FUNCTION_BLOCK Ref_ramp
VAR_INPUT
	Speed_req:INT;
	Allowed_speed:INT;
	Rate:INT;
	Zero:BOOL;
	S_Func_scans:INT;
END_VAR
VAR_OUTPUT
	Speed_ref:INT;
END_VAR
VAR
	Speed_req_real: REAL;
	Speed_step: REAL;
	Speed_ref_real: REAL;
	Speed_up: BOOL;
END_VAR
VAR // added by the converter: edge detectors and wires of the graphical bodies
    _w1, _w2, _w4, _w5, _w6, _w7, _w9, _w10 : ANY;
    _w3 : BOOL;
    _w8, _w11, _w12 : REAL;
END_VAR

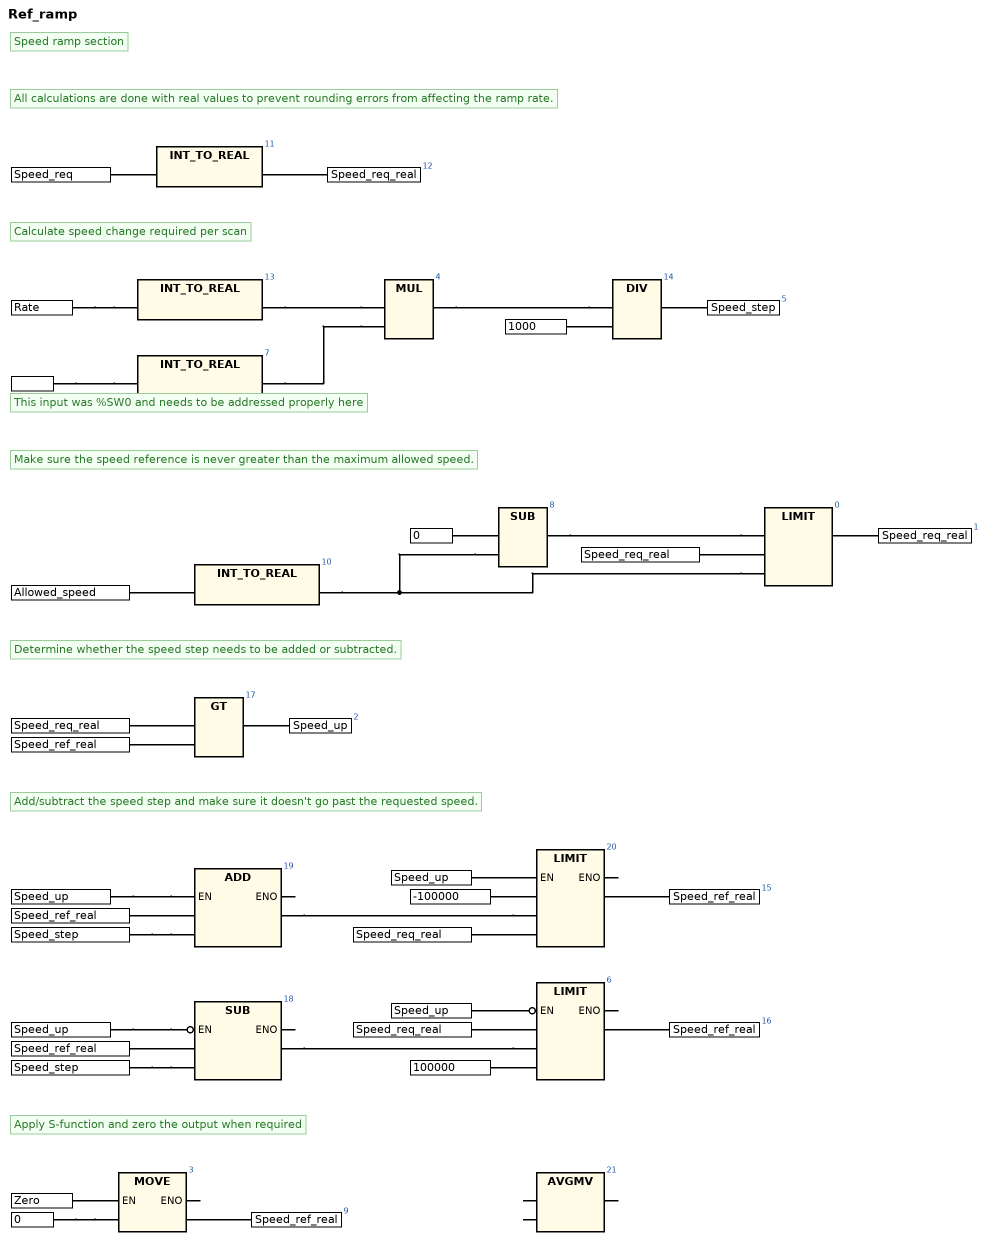
Speed_req_real := LIMIT(_w1, Speed_req_real, _w2);
Speed_up := _w3;
// Apply S-function and zero the output when required
IF Zero THEN _w4 := 0; END_IF
_w7 := _w5 * _w6;
Speed_step := _w8;
IF NOT Speed_up THEN _w10 := LIMIT(Speed_req_real, _w9, 100000); END_IF
// This input was %SW0 and needs to be addressed properly here
_w6 := INT_TO_REAL(???);
_w1 := 0 - _w2;
Speed_ref_real := _w4;
// Make sure the speed reference is never greater than the maximum allowed speed.
_w2 := INT_TO_REAL(Allowed_speed);
// Speed ramp section
// All calculations are done with real values to prevent rounding errors from affecting the ramp rate.
Speed_req_real := INT_TO_REAL(Speed_req);
// Calculate speed change required per scan
_w5 := INT_TO_REAL(Rate);
_w8 := _w7 / 1000;
Speed_ref_real := _w11;
Speed_ref_real := _w10;
// Determine whether the speed step needs to be added or subtracted.
_w3 := Speed_req_real > Speed_ref_real;
IF NOT Speed_up THEN _w9 := Speed_ref_real - Speed_step; END_IF
// Add/subtract the speed step and make sure it doesn't go past the requested speed.
IF Speed_up THEN _w12 := Speed_ref_real + Speed_step; END_IF
IF Speed_up THEN _w11 := LIMIT(-100000, _w12, Speed_req_real); END_IF
AVGMV(???, ???);

END_FUNCTION_BLOCK

(* stored: Version 1.1.0.1, ProductVersion 3.1.4024.0
   POU Ref_ramp: Id {608e08de-3205-4600-9ab4-8b35700b6efb}, SpecialFunc None *)
